(* Logix 5000 project; controller R1USB70001_CWRU_Scenario_Gen_20111116 vendor 1 type 14 code 54 rev 19.11; software revision 19.01; part 8 of 9 *)
(* tags used below, declared in another part *)
   ExecutePv : ExecutePv;
   HMIPv : HMIPv;
   ControlMode : ControlModePub;
   EditScenario : EditScenarioPub;
   Execute : ExecutePub;
   HMI : HMIPub;
   HMI_Intfc_Read_Buffer : DINT[40];
   HMI_Intfc_String_Read_Buffer : STRING[2];
   HMI_Intfc_String_Write_Buffer : STRING;
   HMI_Intfc_Write_Buffer : DINT[20];
(* MainProgram, continued *)

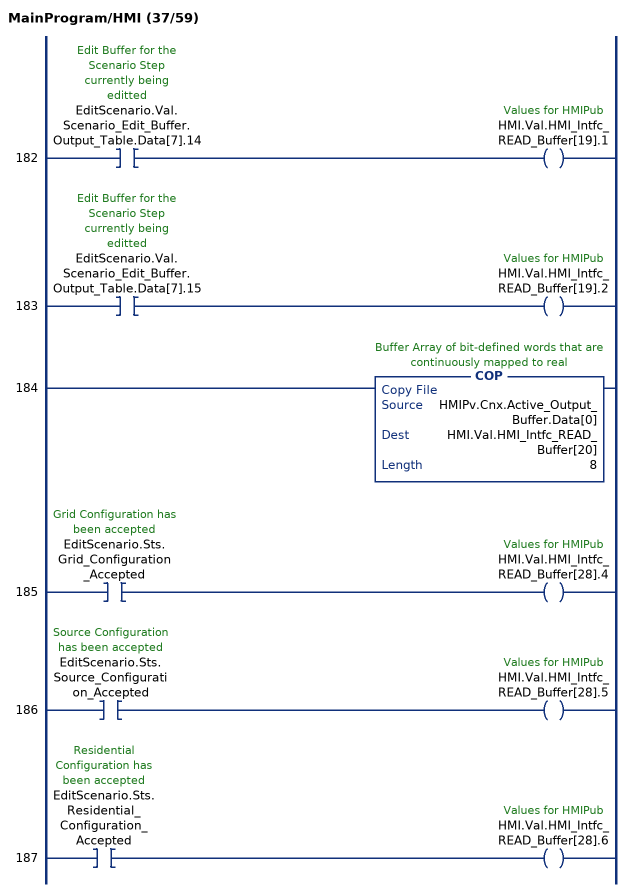
   182: XIC(EditScenario.Val.Scenario_Edit_Buffer.Output_Table.Data[7].14)OTE(HMI.Val.HMI_Intfc_READ_Buffer[19].1);
   183: XIC(EditScenario.Val.Scenario_Edit_Buffer.Output_Table.Data[7].15)OTE(HMI.Val.HMI_Intfc_READ_Buffer[19].2);
   184: COP(HMIPv.Cnx.Active_Output_Buffer.Data[0],HMI.Val.HMI_Intfc_READ_Buffer[20],8);
   185: XIC(EditScenario.Sts.Grid_Configuration_Accepted)OTE(HMI.Val.HMI_Intfc_READ_Buffer[28].4);
   186: XIC(EditScenario.Sts.Source_Configuration_Accepted)OTE(HMI.Val.HMI_Intfc_READ_Buffer[28].5);
   187: XIC(EditScenario.Sts.Residential_Configuration_Accepted)OTE(HMI.Val.HMI_Intfc_READ_Buffer[28].6);
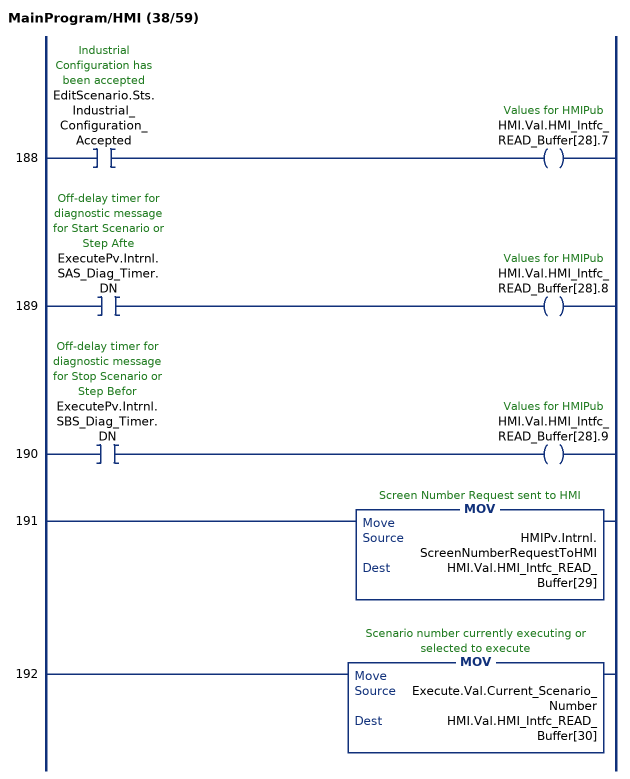
   188: XIC(EditScenario.Sts.Industrial_Configuration_Accepted)OTE(HMI.Val.HMI_Intfc_READ_Buffer[28].7);
   189: XIC(ExecutePv.Intrnl.SAS_Diag_Timer.DN)OTE(HMI.Val.HMI_Intfc_READ_Buffer[28].8);
   190: XIC(ExecutePv.Intrnl.SBS_Diag_Timer.DN)OTE(HMI.Val.HMI_Intfc_READ_Buffer[28].9);
   191: MOV(HMIPv.Intrnl.ScreenNumberRequestToHMI,HMI.Val.HMI_Intfc_READ_Buffer[29]);
   192: MOV(Execute.Val.Current_Scenario_Number,HMI.Val.HMI_Intfc_READ_Buffer[30]);
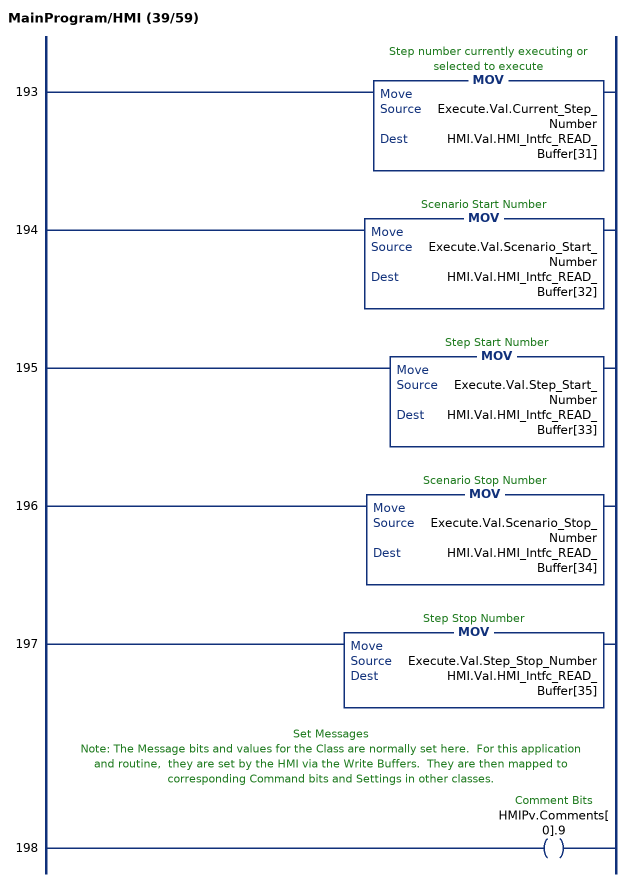
   193: MOV(Execute.Val.Current_Step_Number,HMI.Val.HMI_Intfc_READ_Buffer[31]);
   194: MOV(Execute.Val.Scenario_Start_Number,HMI.Val.HMI_Intfc_READ_Buffer[32]);
   195: MOV(Execute.Val.Step_Start_Number,HMI.Val.HMI_Intfc_READ_Buffer[33]);
   196: MOV(Execute.Val.Scenario_Stop_Number,HMI.Val.HMI_Intfc_READ_Buffer[34]);
   197: MOV(Execute.Val.Step_Stop_Number,HMI.Val.HMI_Intfc_READ_Buffer[35]);
   // Set Messages
   // Note: The Message bits and values for the Class are normally set here.  For this application and routine,  they are set by the HMI via the Write Buffers.  They are then mapped to corresponding Command bits and Settings in other classes.
   198: OTE(HMIPv.Comments[0].9);
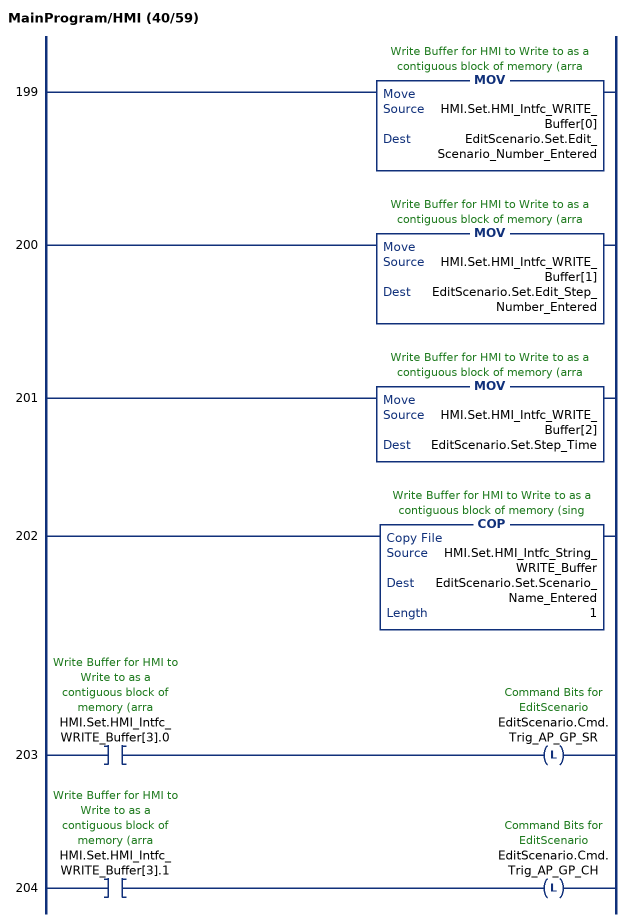
   199: MOV(HMI.Set.HMI_Intfc_WRITE_Buffer[0],EditScenario.Set.Edit_Scenario_Number_Entered);
   200: MOV(HMI.Set.HMI_Intfc_WRITE_Buffer[1],EditScenario.Set.Edit_Step_Number_Entered);
   201: MOV(HMI.Set.HMI_Intfc_WRITE_Buffer[2],EditScenario.Set.Step_Time);
   202: COP(HMI.Set.HMI_Intfc_String_WRITE_Buffer,EditScenario.Set.Scenario_Name_Entered,1);
   203: XIC(HMI.Set.HMI_Intfc_WRITE_Buffer[3].0)OTL(EditScenario.Cmd.Trig_AP_GP_SR);
   204: XIC(HMI.Set.HMI_Intfc_WRITE_Buffer[3].1)OTL(EditScenario.Cmd.Trig_AP_GP_CH);
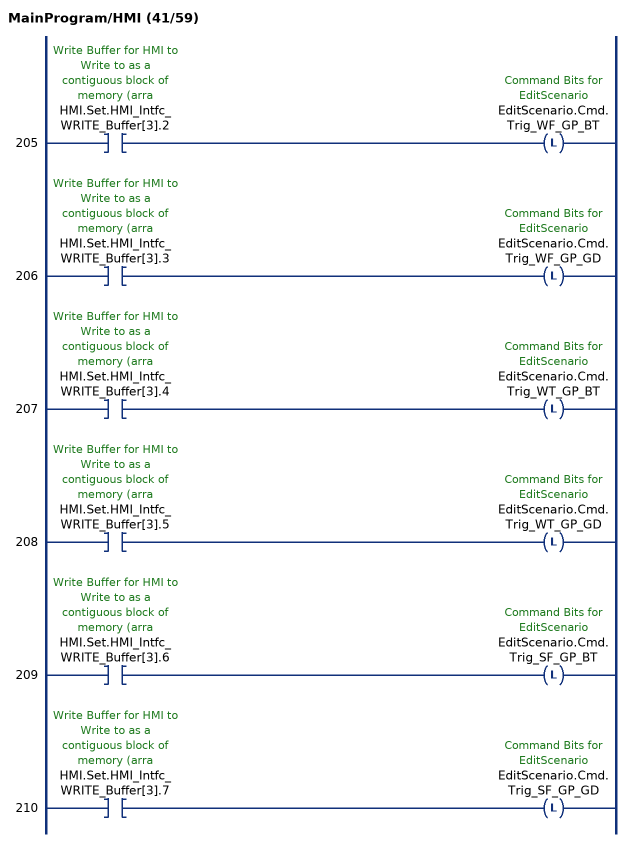
   205: XIC(HMI.Set.HMI_Intfc_WRITE_Buffer[3].2)OTL(EditScenario.Cmd.Trig_WF_GP_BT);
   206: XIC(HMI.Set.HMI_Intfc_WRITE_Buffer[3].3)OTL(EditScenario.Cmd.Trig_WF_GP_GD);
   207: XIC(HMI.Set.HMI_Intfc_WRITE_Buffer[3].4)OTL(EditScenario.Cmd.Trig_WT_GP_BT);
   208: XIC(HMI.Set.HMI_Intfc_WRITE_Buffer[3].5)OTL(EditScenario.Cmd.Trig_WT_GP_GD);
   209: XIC(HMI.Set.HMI_Intfc_WRITE_Buffer[3].6)OTL(EditScenario.Cmd.Trig_SF_GP_BT);
   210: XIC(HMI.Set.HMI_Intfc_WRITE_Buffer[3].7)OTL(EditScenario.Cmd.Trig_SF_GP_GD);
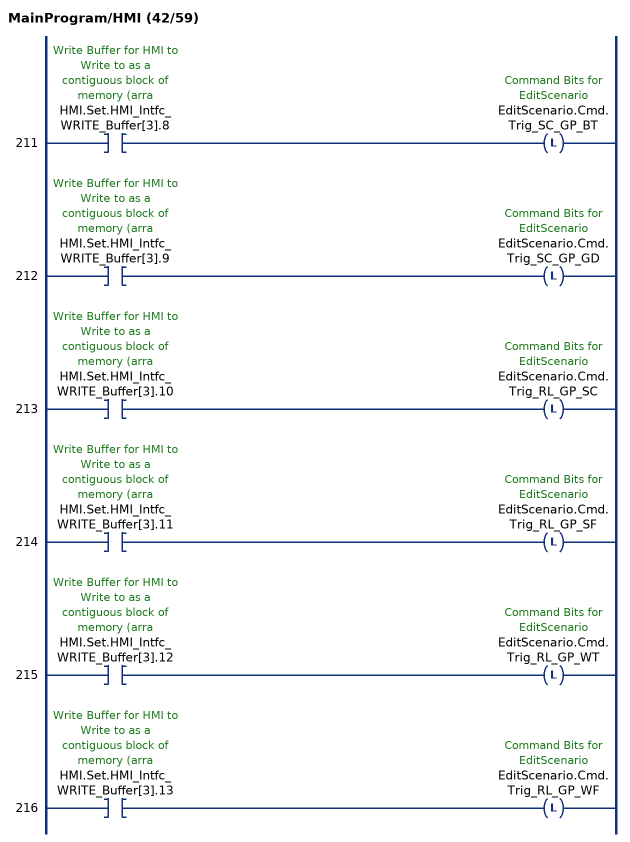
   211: XIC(HMI.Set.HMI_Intfc_WRITE_Buffer[3].8)OTL(EditScenario.Cmd.Trig_SC_GP_BT);
   212: XIC(HMI.Set.HMI_Intfc_WRITE_Buffer[3].9)OTL(EditScenario.Cmd.Trig_SC_GP_GD);
   213: XIC(HMI.Set.HMI_Intfc_WRITE_Buffer[3].10)OTL(EditScenario.Cmd.Trig_RL_GP_SC);
   214: XIC(HMI.Set.HMI_Intfc_WRITE_Buffer[3].11)OTL(EditScenario.Cmd.Trig_RL_GP_SF);
   215: XIC(HMI.Set.HMI_Intfc_WRITE_Buffer[3].12)OTL(EditScenario.Cmd.Trig_RL_GP_WT);
   216: XIC(HMI.Set.HMI_Intfc_WRITE_Buffer[3].13)OTL(EditScenario.Cmd.Trig_RL_GP_WF);
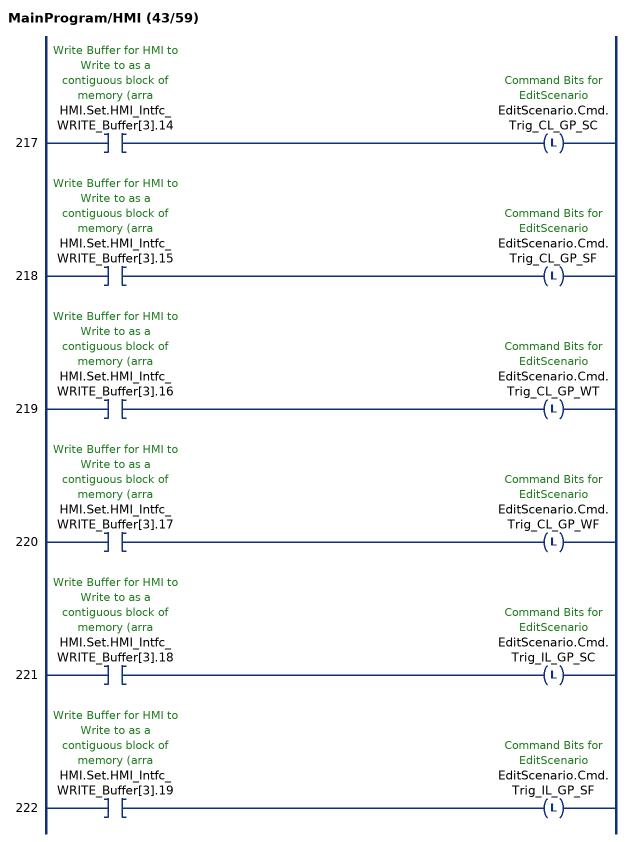
   217: XIC(HMI.Set.HMI_Intfc_WRITE_Buffer[3].14)OTL(EditScenario.Cmd.Trig_CL_GP_SC);
   218: XIC(HMI.Set.HMI_Intfc_WRITE_Buffer[3].15)OTL(EditScenario.Cmd.Trig_CL_GP_SF);
   219: XIC(HMI.Set.HMI_Intfc_WRITE_Buffer[3].16)OTL(EditScenario.Cmd.Trig_CL_GP_WT);
   220: XIC(HMI.Set.HMI_Intfc_WRITE_Buffer[3].17)OTL(EditScenario.Cmd.Trig_CL_GP_WF);
   221: XIC(HMI.Set.HMI_Intfc_WRITE_Buffer[3].18)OTL(EditScenario.Cmd.Trig_IL_GP_SC);
   222: XIC(HMI.Set.HMI_Intfc_WRITE_Buffer[3].19)OTL(EditScenario.Cmd.Trig_IL_GP_SF);
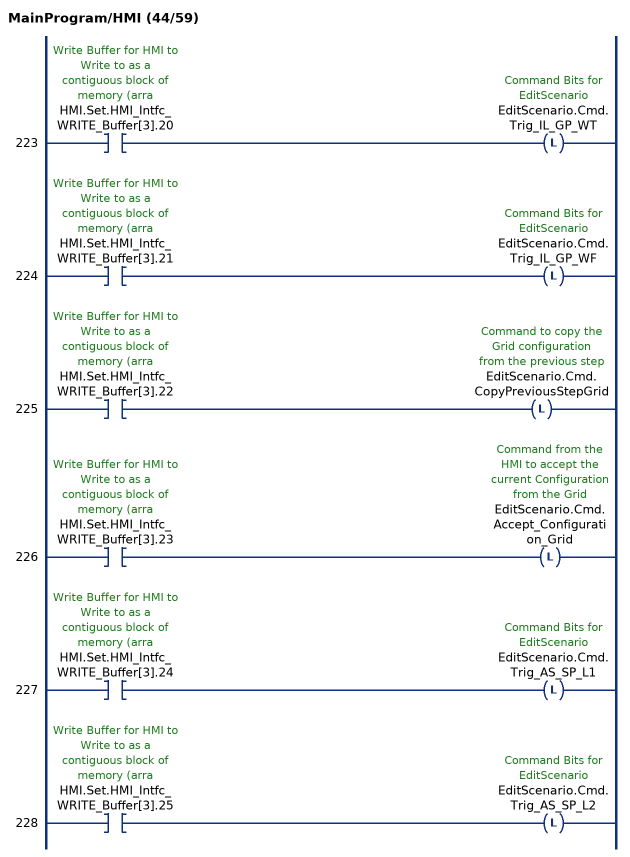
   223: XIC(HMI.Set.HMI_Intfc_WRITE_Buffer[3].20)OTL(EditScenario.Cmd.Trig_IL_GP_WT);
   224: XIC(HMI.Set.HMI_Intfc_WRITE_Buffer[3].21)OTL(EditScenario.Cmd.Trig_IL_GP_WF);
   225: XIC(HMI.Set.HMI_Intfc_WRITE_Buffer[3].22)OTL(EditScenario.Cmd.CopyPreviousStepGrid);
   226: XIC(HMI.Set.HMI_Intfc_WRITE_Buffer[3].23)OTL(EditScenario.Cmd.Accept_Configuration_Grid);
   227: XIC(HMI.Set.HMI_Intfc_WRITE_Buffer[3].24)OTL(EditScenario.Cmd.Trig_AS_SP_L1);
   228: XIC(HMI.Set.HMI_Intfc_WRITE_Buffer[3].25)OTL(EditScenario.Cmd.Trig_AS_SP_L2);
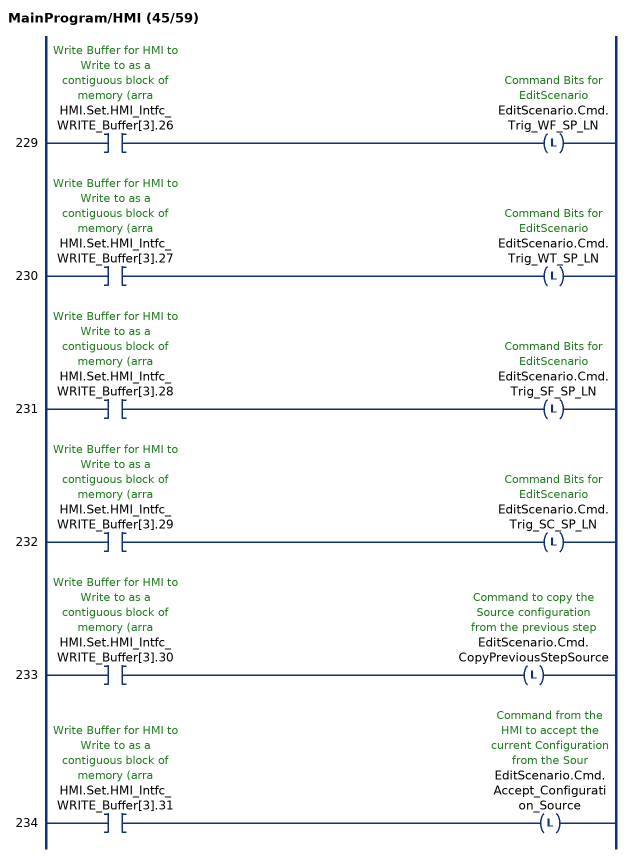
   229: XIC(HMI.Set.HMI_Intfc_WRITE_Buffer[3].26)OTL(EditScenario.Cmd.Trig_WF_SP_LN);
   230: XIC(HMI.Set.HMI_Intfc_WRITE_Buffer[3].27)OTL(EditScenario.Cmd.Trig_WT_SP_LN);
   231: XIC(HMI.Set.HMI_Intfc_WRITE_Buffer[3].28)OTL(EditScenario.Cmd.Trig_SF_SP_LN);
   232: XIC(HMI.Set.HMI_Intfc_WRITE_Buffer[3].29)OTL(EditScenario.Cmd.Trig_SC_SP_LN);
   233: XIC(HMI.Set.HMI_Intfc_WRITE_Buffer[3].30)OTL(EditScenario.Cmd.CopyPreviousStepSource);
   234: XIC(HMI.Set.HMI_Intfc_WRITE_Buffer[3].31)OTL(EditScenario.Cmd.Accept_Configuration_Source);
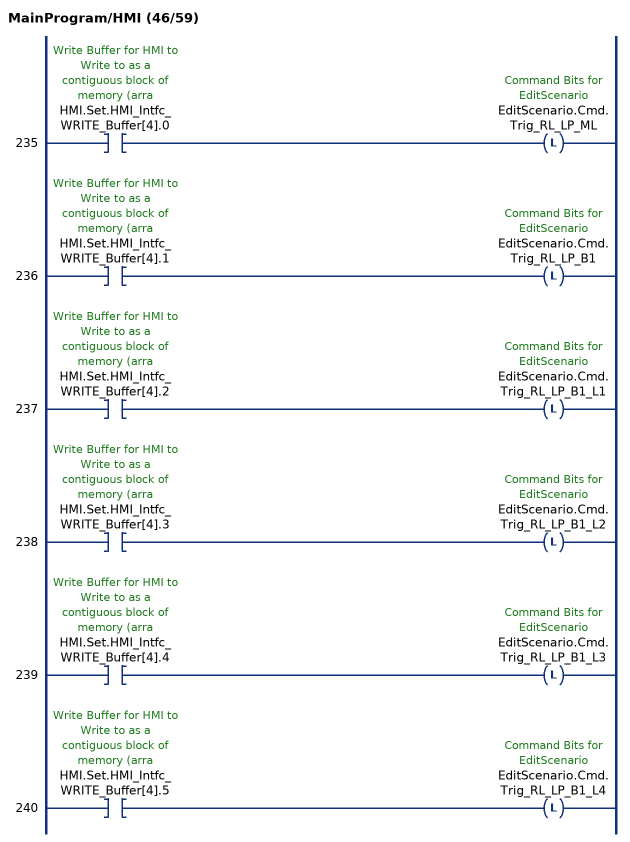
   235: XIC(HMI.Set.HMI_Intfc_WRITE_Buffer[4].0)OTL(EditScenario.Cmd.Trig_RL_LP_ML);
   236: XIC(HMI.Set.HMI_Intfc_WRITE_Buffer[4].1)OTL(EditScenario.Cmd.Trig_RL_LP_B1);
   237: XIC(HMI.Set.HMI_Intfc_WRITE_Buffer[4].2)OTL(EditScenario.Cmd.Trig_RL_LP_B1_L1);
   238: XIC(HMI.Set.HMI_Intfc_WRITE_Buffer[4].3)OTL(EditScenario.Cmd.Trig_RL_LP_B1_L2);
   239: XIC(HMI.Set.HMI_Intfc_WRITE_Buffer[4].4)OTL(EditScenario.Cmd.Trig_RL_LP_B1_L3);
   240: XIC(HMI.Set.HMI_Intfc_WRITE_Buffer[4].5)OTL(EditScenario.Cmd.Trig_RL_LP_B1_L4);
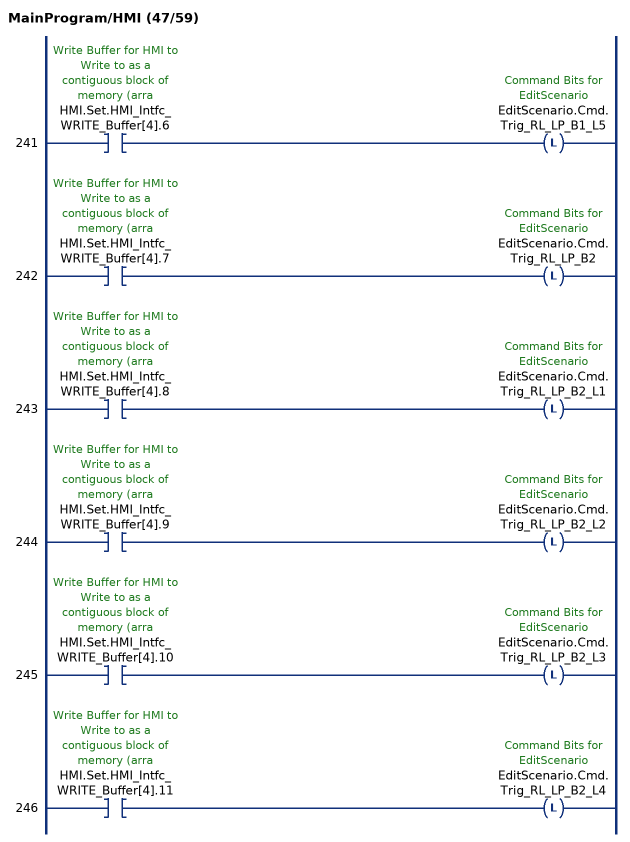
   241: XIC(HMI.Set.HMI_Intfc_WRITE_Buffer[4].6)OTL(EditScenario.Cmd.Trig_RL_LP_B1_L5);
   242: XIC(HMI.Set.HMI_Intfc_WRITE_Buffer[4].7)OTL(EditScenario.Cmd.Trig_RL_LP_B2);
   243: XIC(HMI.Set.HMI_Intfc_WRITE_Buffer[4].8)OTL(EditScenario.Cmd.Trig_RL_LP_B2_L1);
   244: XIC(HMI.Set.HMI_Intfc_WRITE_Buffer[4].9)OTL(EditScenario.Cmd.Trig_RL_LP_B2_L2);
   245: XIC(HMI.Set.HMI_Intfc_WRITE_Buffer[4].10)OTL(EditScenario.Cmd.Trig_RL_LP_B2_L3);
   246: XIC(HMI.Set.HMI_Intfc_WRITE_Buffer[4].11)OTL(EditScenario.Cmd.Trig_RL_LP_B2_L4);
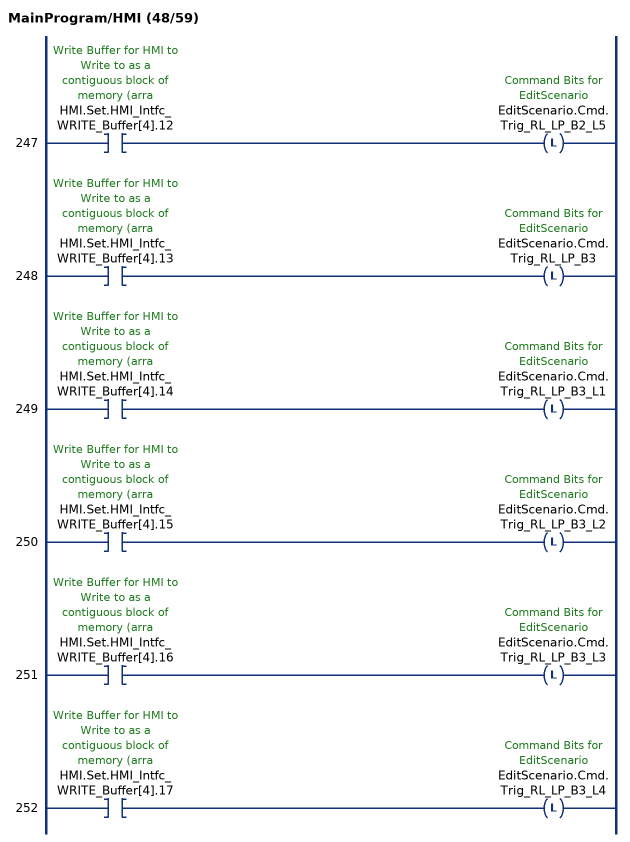
   247: XIC(HMI.Set.HMI_Intfc_WRITE_Buffer[4].12)OTL(EditScenario.Cmd.Trig_RL_LP_B2_L5);
   248: XIC(HMI.Set.HMI_Intfc_WRITE_Buffer[4].13)OTL(EditScenario.Cmd.Trig_RL_LP_B3);
   249: XIC(HMI.Set.HMI_Intfc_WRITE_Buffer[4].14)OTL(EditScenario.Cmd.Trig_RL_LP_B3_L1);
   250: XIC(HMI.Set.HMI_Intfc_WRITE_Buffer[4].15)OTL(EditScenario.Cmd.Trig_RL_LP_B3_L2);
   251: XIC(HMI.Set.HMI_Intfc_WRITE_Buffer[4].16)OTL(EditScenario.Cmd.Trig_RL_LP_B3_L3);
   252: XIC(HMI.Set.HMI_Intfc_WRITE_Buffer[4].17)OTL(EditScenario.Cmd.Trig_RL_LP_B3_L4);
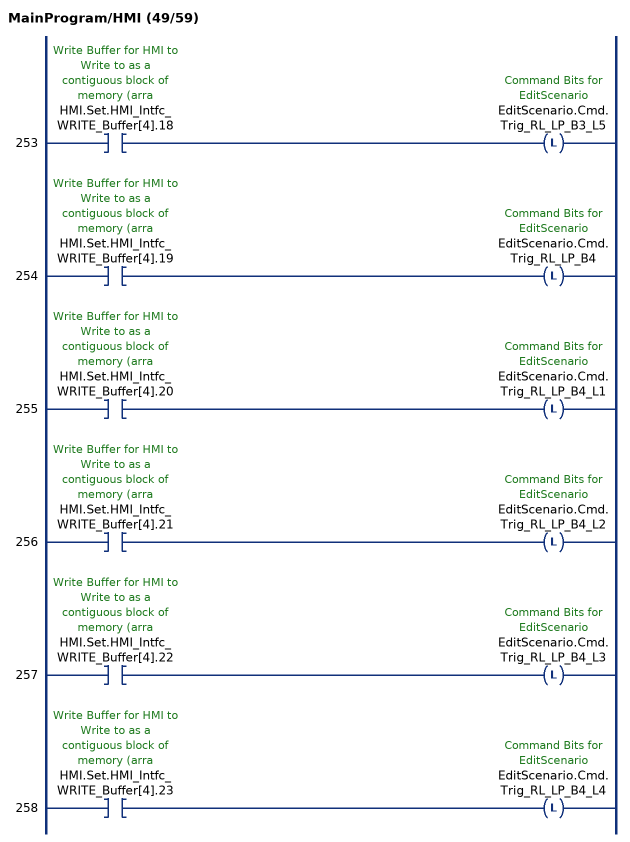
   253: XIC(HMI.Set.HMI_Intfc_WRITE_Buffer[4].18)OTL(EditScenario.Cmd.Trig_RL_LP_B3_L5);
   254: XIC(HMI.Set.HMI_Intfc_WRITE_Buffer[4].19)OTL(EditScenario.Cmd.Trig_RL_LP_B4);
   255: XIC(HMI.Set.HMI_Intfc_WRITE_Buffer[4].20)OTL(EditScenario.Cmd.Trig_RL_LP_B4_L1);
   256: XIC(HMI.Set.HMI_Intfc_WRITE_Buffer[4].21)OTL(EditScenario.Cmd.Trig_RL_LP_B4_L2);
   257: XIC(HMI.Set.HMI_Intfc_WRITE_Buffer[4].22)OTL(EditScenario.Cmd.Trig_RL_LP_B4_L3);
   258: XIC(HMI.Set.HMI_Intfc_WRITE_Buffer[4].23)OTL(EditScenario.Cmd.Trig_RL_LP_B4_L4);
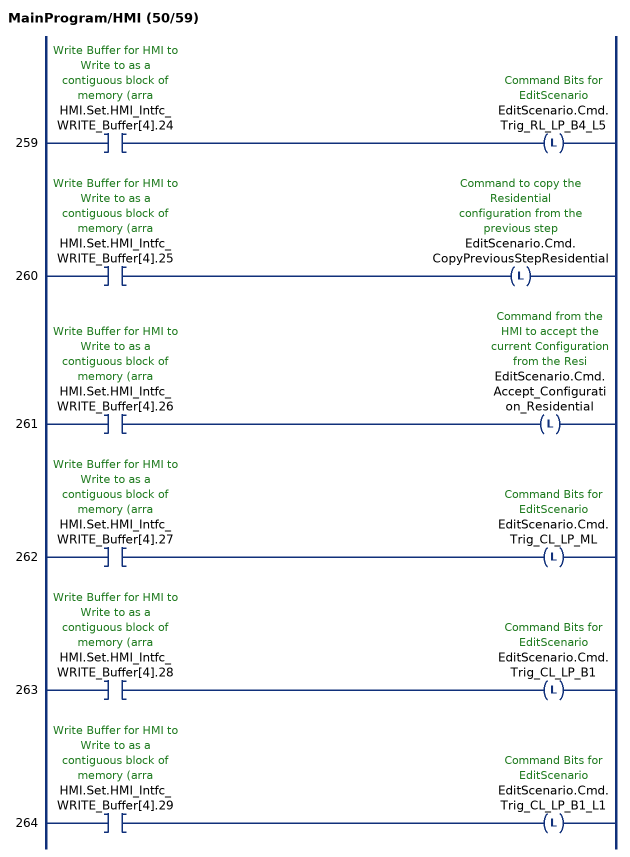
   259: XIC(HMI.Set.HMI_Intfc_WRITE_Buffer[4].24)OTL(EditScenario.Cmd.Trig_RL_LP_B4_L5);
   260: XIC(HMI.Set.HMI_Intfc_WRITE_Buffer[4].25)OTL(EditScenario.Cmd.CopyPreviousStepResidential);
   261: XIC(HMI.Set.HMI_Intfc_WRITE_Buffer[4].26)OTL(EditScenario.Cmd.Accept_Configuration_Residential);
   262: XIC(HMI.Set.HMI_Intfc_WRITE_Buffer[4].27)OTL(EditScenario.Cmd.Trig_CL_LP_ML);
   263: XIC(HMI.Set.HMI_Intfc_WRITE_Buffer[4].28)OTL(EditScenario.Cmd.Trig_CL_LP_B1);
   264: XIC(HMI.Set.HMI_Intfc_WRITE_Buffer[4].29)OTL(EditScenario.Cmd.Trig_CL_LP_B1_L1);
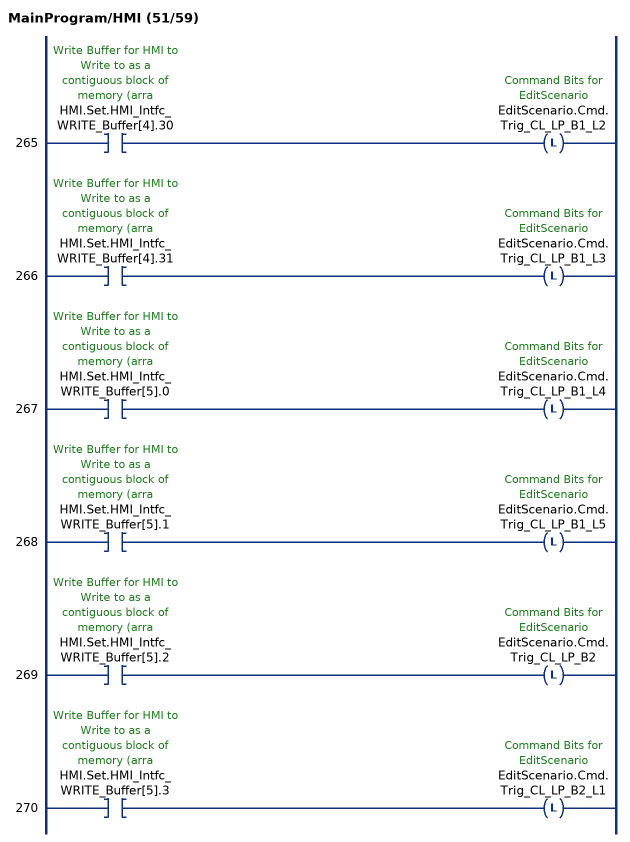
   265: XIC(HMI.Set.HMI_Intfc_WRITE_Buffer[4].30)OTL(EditScenario.Cmd.Trig_CL_LP_B1_L2);
   266: XIC(HMI.Set.HMI_Intfc_WRITE_Buffer[4].31)OTL(EditScenario.Cmd.Trig_CL_LP_B1_L3);
   267: XIC(HMI.Set.HMI_Intfc_WRITE_Buffer[5].0)OTL(EditScenario.Cmd.Trig_CL_LP_B1_L4);
   268: XIC(HMI.Set.HMI_Intfc_WRITE_Buffer[5].1)OTL(EditScenario.Cmd.Trig_CL_LP_B1_L5);
   269: XIC(HMI.Set.HMI_Intfc_WRITE_Buffer[5].2)OTL(EditScenario.Cmd.Trig_CL_LP_B2);
   270: XIC(HMI.Set.HMI_Intfc_WRITE_Buffer[5].3)OTL(EditScenario.Cmd.Trig_CL_LP_B2_L1);
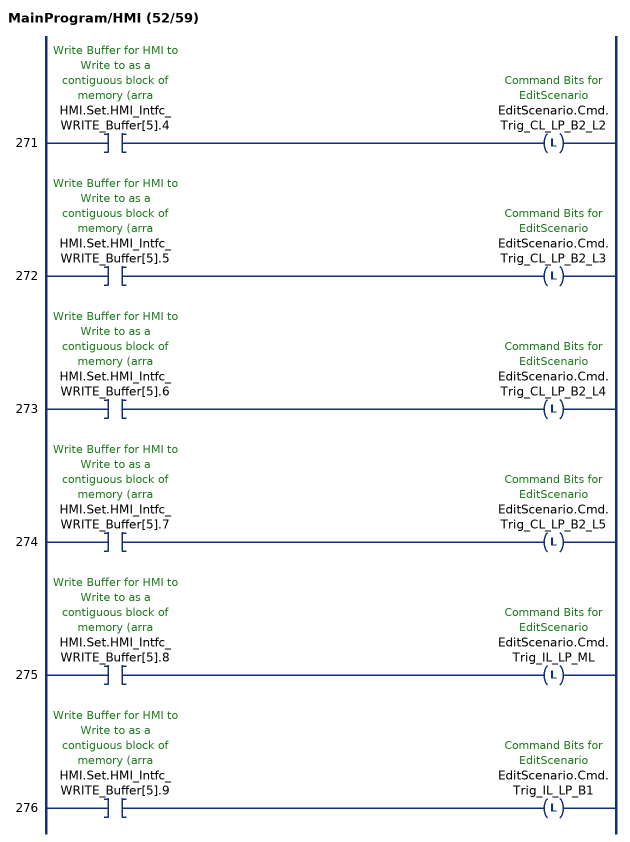
   271: XIC(HMI.Set.HMI_Intfc_WRITE_Buffer[5].4)OTL(EditScenario.Cmd.Trig_CL_LP_B2_L2);
   272: XIC(HMI.Set.HMI_Intfc_WRITE_Buffer[5].5)OTL(EditScenario.Cmd.Trig_CL_LP_B2_L3);
   273: XIC(HMI.Set.HMI_Intfc_WRITE_Buffer[5].6)OTL(EditScenario.Cmd.Trig_CL_LP_B2_L4);
   274: XIC(HMI.Set.HMI_Intfc_WRITE_Buffer[5].7)OTL(EditScenario.Cmd.Trig_CL_LP_B2_L5);
   275: XIC(HMI.Set.HMI_Intfc_WRITE_Buffer[5].8)OTL(EditScenario.Cmd.Trig_IL_LP_ML);
   276: XIC(HMI.Set.HMI_Intfc_WRITE_Buffer[5].9)OTL(EditScenario.Cmd.Trig_IL_LP_B1);
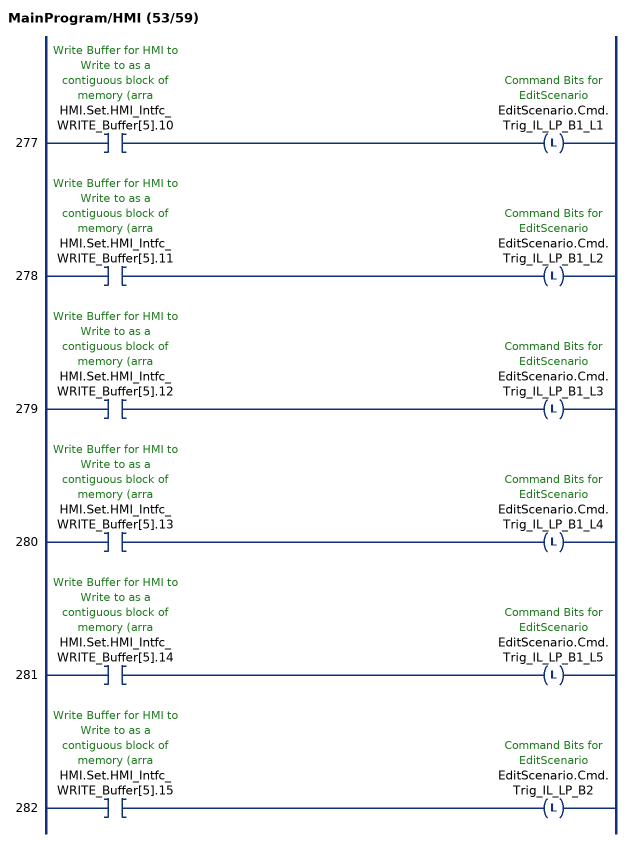
   277: XIC(HMI.Set.HMI_Intfc_WRITE_Buffer[5].10)OTL(EditScenario.Cmd.Trig_IL_LP_B1_L1);
   278: XIC(HMI.Set.HMI_Intfc_WRITE_Buffer[5].11)OTL(EditScenario.Cmd.Trig_IL_LP_B1_L2);
   279: XIC(HMI.Set.HMI_Intfc_WRITE_Buffer[5].12)OTL(EditScenario.Cmd.Trig_IL_LP_B1_L3);
   280: XIC(HMI.Set.HMI_Intfc_WRITE_Buffer[5].13)OTL(EditScenario.Cmd.Trig_IL_LP_B1_L4);
   281: XIC(HMI.Set.HMI_Intfc_WRITE_Buffer[5].14)OTL(EditScenario.Cmd.Trig_IL_LP_B1_L5);
   282: XIC(HMI.Set.HMI_Intfc_WRITE_Buffer[5].15)OTL(EditScenario.Cmd.Trig_IL_LP_B2);
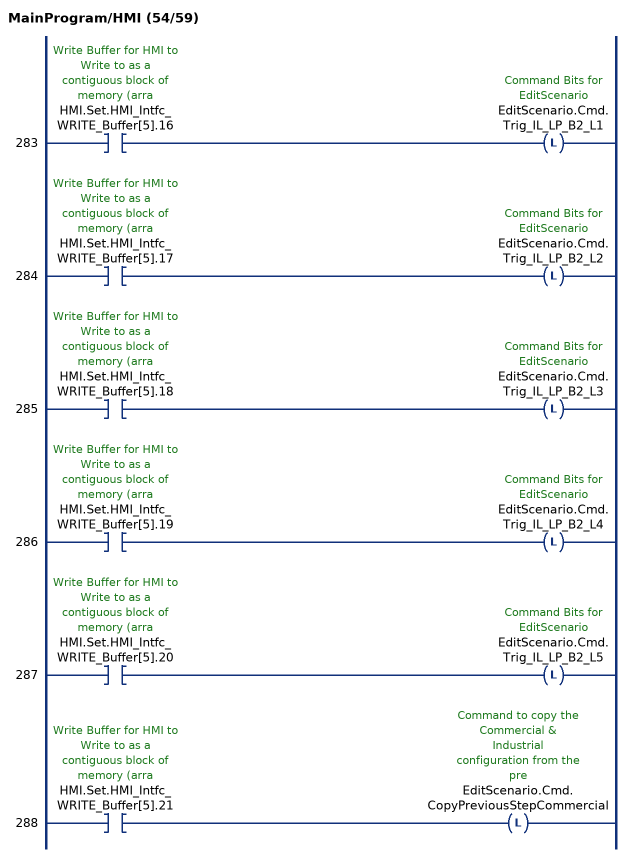
   283: XIC(HMI.Set.HMI_Intfc_WRITE_Buffer[5].16)OTL(EditScenario.Cmd.Trig_IL_LP_B2_L1);
   284: XIC(HMI.Set.HMI_Intfc_WRITE_Buffer[5].17)OTL(EditScenario.Cmd.Trig_IL_LP_B2_L2);
   285: XIC(HMI.Set.HMI_Intfc_WRITE_Buffer[5].18)OTL(EditScenario.Cmd.Trig_IL_LP_B2_L3);
   286: XIC(HMI.Set.HMI_Intfc_WRITE_Buffer[5].19)OTL(EditScenario.Cmd.Trig_IL_LP_B2_L4);
   287: XIC(HMI.Set.HMI_Intfc_WRITE_Buffer[5].20)OTL(EditScenario.Cmd.Trig_IL_LP_B2_L5);
   288: XIC(HMI.Set.HMI_Intfc_WRITE_Buffer[5].21)OTL(EditScenario.Cmd.CopyPreviousStepCommercial);
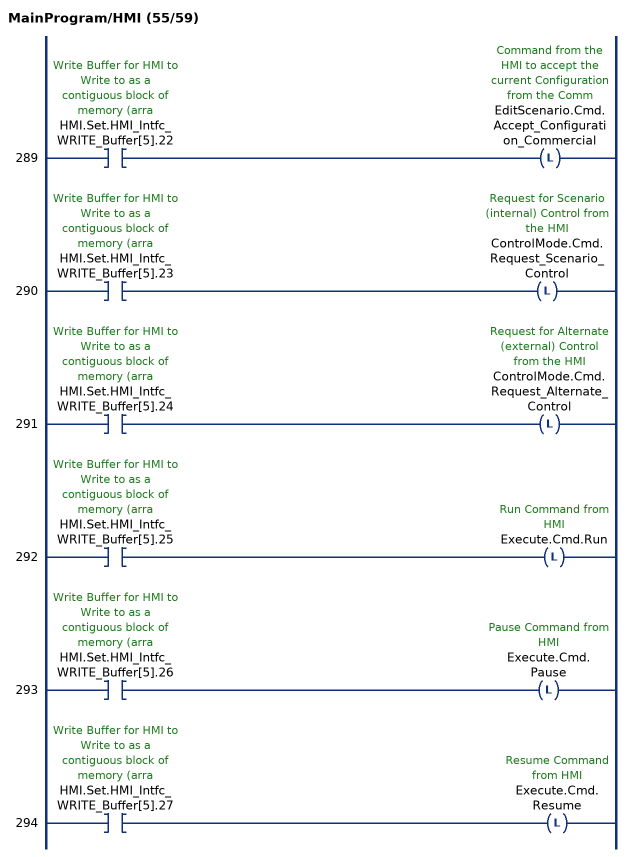
   289: XIC(HMI.Set.HMI_Intfc_WRITE_Buffer[5].22)OTL(EditScenario.Cmd.Accept_Configuration_Commercial);
   290: XIC(HMI.Set.HMI_Intfc_WRITE_Buffer[5].23)OTL(ControlMode.Cmd.Request_Scenario_Control);
   291: XIC(HMI.Set.HMI_Intfc_WRITE_Buffer[5].24)OTL(ControlMode.Cmd.Request_Alternate_Control);
   292: XIC(HMI.Set.HMI_Intfc_WRITE_Buffer[5].25)OTL(Execute.Cmd.Run);
   293: XIC(HMI.Set.HMI_Intfc_WRITE_Buffer[5].26)OTL(Execute.Cmd.Pause);
   294: XIC(HMI.Set.HMI_Intfc_WRITE_Buffer[5].27)OTL(Execute.Cmd.Resume);
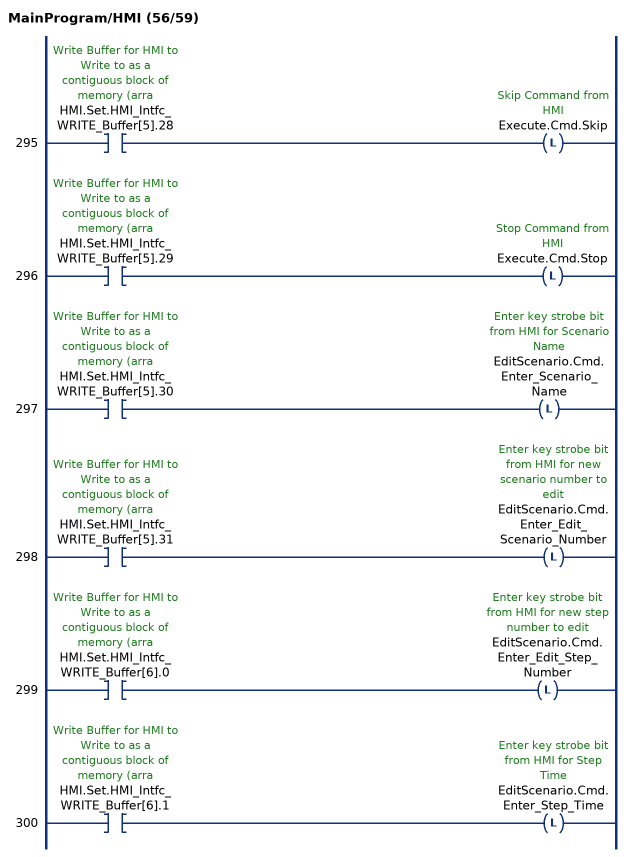
   295: XIC(HMI.Set.HMI_Intfc_WRITE_Buffer[5].28)OTL(Execute.Cmd.Skip);
   296: XIC(HMI.Set.HMI_Intfc_WRITE_Buffer[5].29)OTL(Execute.Cmd.Stop);
   297: XIC(HMI.Set.HMI_Intfc_WRITE_Buffer[5].30)OTL(EditScenario.Cmd.Enter_Scenario_Name);
   298: XIC(HMI.Set.HMI_Intfc_WRITE_Buffer[5].31)OTL(EditScenario.Cmd.Enter_Edit_Scenario_Number);
   299: XIC(HMI.Set.HMI_Intfc_WRITE_Buffer[6].0)OTL(EditScenario.Cmd.Enter_Edit_Step_Number);
   300: XIC(HMI.Set.HMI_Intfc_WRITE_Buffer[6].1)OTL(EditScenario.Cmd.Enter_Step_Time);
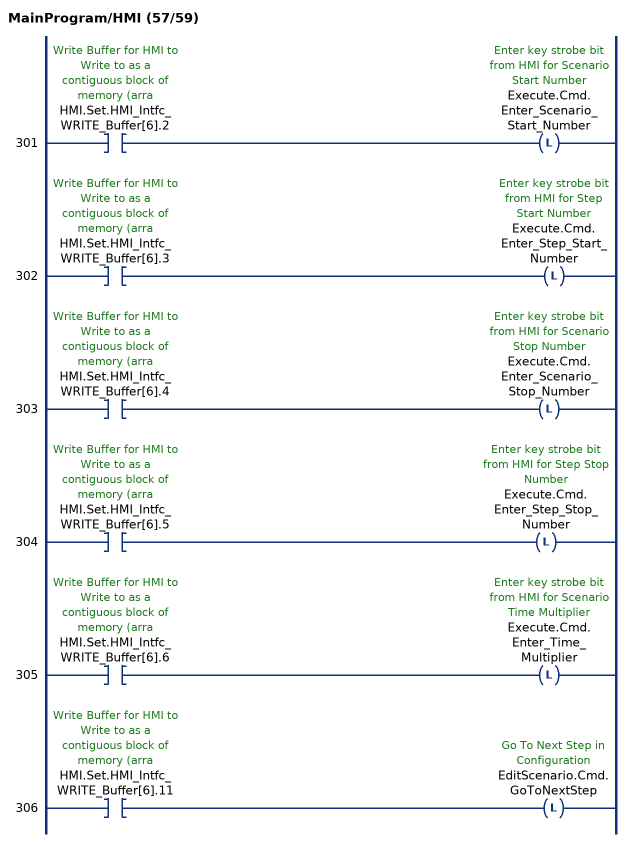
   301: XIC(HMI.Set.HMI_Intfc_WRITE_Buffer[6].2)OTL(Execute.Cmd.Enter_Scenario_Start_Number);
   302: XIC(HMI.Set.HMI_Intfc_WRITE_Buffer[6].3)OTL(Execute.Cmd.Enter_Step_Start_Number);
   303: XIC(HMI.Set.HMI_Intfc_WRITE_Buffer[6].4)OTL(Execute.Cmd.Enter_Scenario_Stop_Number);
   304: XIC(HMI.Set.HMI_Intfc_WRITE_Buffer[6].5)OTL(Execute.Cmd.Enter_Step_Stop_Number);
   305: XIC(HMI.Set.HMI_Intfc_WRITE_Buffer[6].6)OTL(Execute.Cmd.Enter_Time_Multiplier);
   306: XIC(HMI.Set.HMI_Intfc_WRITE_Buffer[6].11)OTL(EditScenario.Cmd.GoToNextStep);
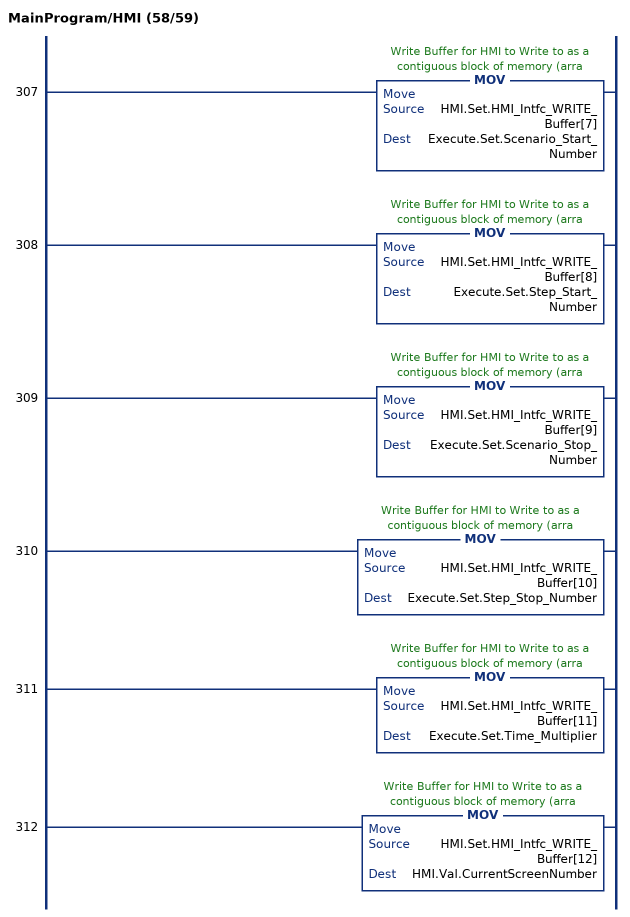
   307: MOV(HMI.Set.HMI_Intfc_WRITE_Buffer[7],Execute.Set.Scenario_Start_Number);
   308: MOV(HMI.Set.HMI_Intfc_WRITE_Buffer[8],Execute.Set.Step_Start_Number);
   309: MOV(HMI.Set.HMI_Intfc_WRITE_Buffer[9],Execute.Set.Scenario_Stop_Number);
   310: MOV(HMI.Set.HMI_Intfc_WRITE_Buffer[10],Execute.Set.Step_Stop_Number);
   311: MOV(HMI.Set.HMI_Intfc_WRITE_Buffer[11],Execute.Set.Time_Multiplier);
   312: MOV(HMI.Set.HMI_Intfc_WRITE_Buffer[12],HMI.Val.CurrentScreenNumber);
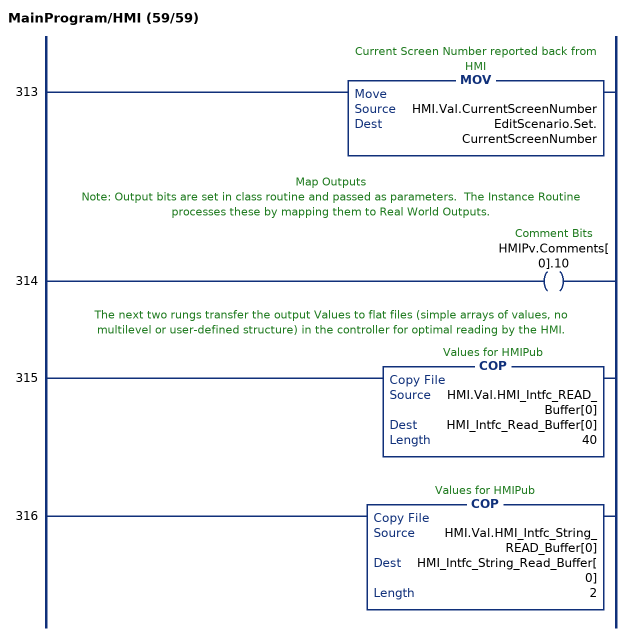
   313: MOV(HMI.Val.CurrentScreenNumber,EditScenario.Set.CurrentScreenNumber);
   // Map Outputs
   // Note: Output bits are set in class routine and passed as parameters.  The Instance Routine processes these by mapping them to Real World Outputs.
   314: OTE(HMIPv.Comments[0].10);
   // The next two rungs transfer the output Values to flat files (simple arrays of values, no multilevel or user-defined structure) in the controller for optimal reading by the HMI.
   315: COP(HMI.Val.HMI_Intfc_READ_Buffer[0],HMI_Intfc_Read_Buffer[0],40);
   316: COP(HMI.Val.HMI_Intfc_String_READ_Buffer[0],HMI_Intfc_String_Read_Buffer[0],2);
END_ROUTINE
